// Mitsubishi GX Works2 project: 실습1-3동일출력2개스위치   PLC: Q02/Q02H

PROGRAM MAIN
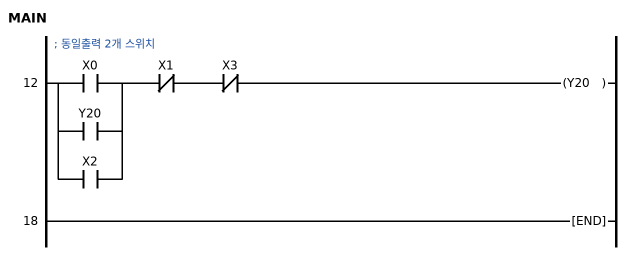
; 동일출력 2개 스위치
12    LD      X0
      OR      Y20
      OR      X2
      ANI     X1
      ANI     X3
      OUT     Y20
18    END
END_PROGRAM
